FUNCTION_BLOCK AdsHandle_1
VAR_OUTPUT
	RemotePrgName		: STRING;
	RemoteNetId			: STRING; 	(* Server AmsNetId *)
	RemotePort 			: UINT;		(* Server port number *)
	
	LocalPrgName 		: STRING;
	LocalNetId 			: STRING;
	LocalPort 			: UINT;
	
	remoteAccessPrefix	: STRING;
	
	busy				: BOOL;
	error					: BOOL;
	errorId				: UDINT;
	
	receiveBuffer		: ARRAY[0..100000] OF BYTE; //TCP style data buffer
	receiveStruct		: AdsData;
END_VAR
VAR
	adsReadSymbol : FB_ReadAdsSymByName;
	adsWriteSymbol : FB_WriteAdsSymByName;
	
	sendQueue			: AdsDataQueue;
	sendBufferQueue 	: DynamicQueue; //anything going into this needs to be a TcpStruct
	
	sendBuffer 			: ARRAY[0..50000] OF BYTE; //temp byte buffer to send if neccessary
	sendStruct			: AdsData;
	
	setupStep 			: (SET_LOCAL_ENDPOINT, CLOSE_CONNECTIONS, SEND_CONNECTION_DATA, RECEIVE_SERVER_DATA, FINISH_SETUP);
	writeDelay : TON;
	
	i : INT;
	adsCtr : INT;
END_VAR
VAR_STAT CONSTANT
	emptyData : AdsData;
	writeDelayTime : TIME := T#1S;
END_VAR

writeDelay(IN:= , PT:= writeDelayTime, Q=> , ET=> );
writeDelay.IN := NOT adsWriteSymbol.bBusy;

blocks();

IF writeDelay.Q THEN
	write();
END_IF

METHOD blocks : BOOL
adsWriteSymbol(
	bWrite:= , 
	sNetId:= RemoteNetId, 
	nPort:= RemotePort, 
	sVarName:= , 
	nSrcAddr:= , 
	nLen:= , 
	tTimeout:= , 
	eComMode:= , 
	bBusy=> , 
	bError=> , 
	nErrorId=> );

adsReadSymbol(
	bRead:= , 
	sNetId:= RemoteNetId, 
	nPort:= RemotePort, 
	sVarName:= , 
	nDestAddr:= , 
	nLen:= , 
	tTimeout:= , 
	eComMode:= , 
	bClearOnError:= TRUE, 
	bBusy=> ,
	bError=> , 
	nErrorId=> );

adsReadSymbol.bRead := NOT adsReadSymbol.bRead;
END_METHOD

METHOD clearBuffer : BOOL
VAR
	emptyReceiverStruct : AdsData;
END_VAR
//MEMSET(ADR(receiveBuffer), 0, SIZEOF(receiveBuffer));
receiveStruct := emptyReceiverStruct;
END_METHOD

METHOD getHandlerName : STRING
getHandlerName := socket.remotePrgName;
END_METHOD

METHOD open : BOOL
VAR_INPUT
	localPrgName : STRING;
	localNetId : T_AmsNetId;
	localPort : T_AmsPort;
END_VAR
socket.open(localPrgName, localNetId, localPort);
END_METHOD

METHOD queueData : BOOL
VAR_INPUT
	data : REFERENCE TO AdsData;
END_VAR
//MEMCPY(ADR(temp), data.pValue, data.diSize);
sendQueue.push(data);
END_METHOD

METHOD read : BOOL
VAR_INPUT
	symbol : STRING;
	buffer : PVOID;
	symbolSize : UDINT;
END_VAR
IF NOT socket.readBusy THEN
	read := socket.read(
		symbol:= symbol,
		buffer := buffer,
		symbolSize := symbolSize);
END_IF
END_METHOD

METHOD PROTECTED setup : BOOL
VAR
	pass : BOOL;
END_VAR
CASE setupStep OF
	SET_LOCAL_ENDPOINT:
		IF
			localPrgName <> '' AND
			localNetId <> '' AND localNetId <> '0.0.0.0.0.0' OR
			localPort <> 0
		THEN
			setupStep := SEND_CONNECTION_DATA;
		END_IF
		
	SEND_CONNECTION_DATA: //send local name, net id, and port
		IF adsWriteSymbol.bWrite AND NOT adsWriteSymbol.bBusy AND NOT adsWriteSymbol.bError THEN //writing done
			adsWriteSymbol.bWrite := FALSE;
			adsCtr := adsCtr + 1;
		END_IF
		
		CASE adsCtr OF
			0:
				adsWriteSymbol.bWrite := NOT adsWriteSymbol.bWrite;
				
				adsWriteSymbol.sVarName := CONCAT(remoteAccessPrefix, 'RemotePrgName');
				adsWriteSymbol.nSrcAddr := ADR(LocalPrgName);
				adsWriteSymbol.nLen := SIZEOF(LocalPrgName);
			
			1:
				
				adsWriteSymbol.bWrite := NOT adsWriteSymbol.bWrite;
				
				adsWriteSymbol.sVarName := CONCAT(remoteAccessPrefix, 'RemoteNetId');
				adsWriteSymbol.nSrcAddr := ADR(LocalNetId);
				adsWriteSymbol.nLen := SIZEOF(LocalNetId);
			
			2:
				
				adsWriteSymbol.bWrite := NOT adsWriteSymbol.bWrite;
				
				adsWriteSymbol.sVarName := CONCAT(remoteAccessPrefix, 'RemotePort');
				adsWriteSymbol.nSrcAddr := ADR(LocalPort);
				adsWriteSymbol.nLen := SIZEOF(LocalPort);
			
			3:
				adsCtr := 0;
				setupStep := RECEIVE_SERVER_DATA;			
		END_CASE
		
	RECEIVE_SERVER_DATA: //get server name, net id and port should already be known
		IF adsReadSymbol.bRead AND NOT adsReadSymbol.bBusy AND NOT adsReadSymbol.bError THEN //reading done
			adsReadSymbol.bRead := FALSE;
			adsCtr := adsCtr + 1;
		END_IF
			
		CASE adsCtr OF
			0:
				adsReadSymbol.bRead := NOT adsReadSymbol.bRead;
				
				adsReadSymbol.sVarName := CONCAT(remoteAccessPrefix, 'LocalPrgName');
				adsReadSymbol.nDestAddr := ADR(RemotePrgName);
				adsReadSymbol.nLen := SIZEOF(RemotePrgName);
			
			1:
				adsReadSymbol.bRead := NOT adsReadSymbol.bRead;
				
				adsReadSymbol.sVarName := CONCAT(remoteAccessPrefix, 'LocalNetId');
				adsReadSymbol.nDestAddr := ADR(RemoteNetId);
				adsReadSymbol.nLen := SIZEOF(RemoteNetId);
			
			2:
				adsReadSymbol.bRead := NOT adsReadSymbol.bRead;
				
				adsReadSymbol.sVarName := CONCAT(remoteAccessPrefix, 'LocalPort');
				adsReadSymbol.nDestAddr := ADR(RemotePort);
				adsReadSymbol.nLen := SIZEOF(RemotePort);
			
			3:
				adsCtr := 0;
				setupStep := FINISH_SETUP;
				RETURN;
			
		END_CASE
			
	FINISH_SETUP:
		setup := TRUE;
		RETURN;
END_CASE
END_METHOD

METHOD write : BOOL
sendStruct := sendQueue.poll();
	
IF MEMCMP(ADR(sendStruct), ADR(emptyData), SIZEOF(AdsData)) <> 0 THEN //if valid data to send
	adsWriteSymbol.nSrcAddr := ADR(sendStruct);
	adsWriteSymbol.nSrcAddr := SIZEOF(sendStruct);
	adsWriteSymbol.sVarName := CONCAT(remoteAccessPrefix, 'receiveStruct');
	
ELSE
	adsWriteSymbol.bWrite := FALSE;
	
END_IF
END_METHOD

END_FUNCTION_BLOCK

(* stored: Version 1.1.0.1, ProductVersion 3.1.4024.11
   POU AdsHandle_1: Id {5a218303-dd26-4595-a947-087b58fe398c}, SpecialFunc None
   Folder ADS: Id {5198003b-35fa-40da-b54d-ad55456f1592}
   Method blocks: Id {f052b581-8913-4a0d-aea6-c77278ede5be}
   Method clearBuffer: Id {f22f11dc-561c-4f67-9d1f-a4322f853329}
   Method getHandlerName: Id {cd418a63-b2bf-4855-8fea-fd46b9f0d3ee}
   Method open: Id {bf1b682c-1dab-40dd-a933-95ce80b26f28}
   Method queueData: Id {68707bae-c360-457e-b457-1c68d7ee70fc}
   Method read: Id {d024bde5-4633-4122-9df7-0ed6612e9dd3}
   Method setup: Id {8c0435c7-4c46-40f4-ae10-d4cd941c6aca}
   Method write: Id {3f12e3ed-096b-4596-81da-20a77bb033f8} *)
